FUNCTION FC_GetLocalAmsNetId : T_AmsNetId		// Returns the local AMS net id

FC_GetLocalAmsNetId := IING.localAmsNetId;

END_FUNCTION

(* stored: Version 1.1.0.1, ProductVersion 3.1.4026.18
   POU FC_GetLocalAmsNetId: Id {e51e6130-b7b0-4201-9df8-3a3213a1e5d5}, SpecialFunc None *)
